// TIA Portal project "Projeto Base" (V17)

(* hardware
DEVICE "S7-1200 station_1"  S7-1200 Station
   slot 0: "Rack_0"  S7-1200 Rack  Rack  V1.0
   slot 1: "PLC_1"  CPU 1212C DC/DC/DC  6ES7 212-1AE40-0XB0  V4.4
DEVICE "HMI_2"  TP700 Comfort
   slot 0: "HMI_2"  TP700 Comfort  6AV2 124-0GC01-0AX0  17.0.0.0
   slot 1: "HMI_RT_2"  TP700 Comfort  6AV2 124-0GC01-0AX0  17.0.0.0
   slot 5: "HMI_2.IE_CP_1"  PROFINET Interface  17.0.0.0
      slot 1: "PROFINET Interface_1"  PROFINET Interface
         slot 1: "Port_1"  Port
         slot 2: "Port_2"  Port
   slot 7: "HMI_2.MPI/DP_CP_1"  MPI/DP Interface  17.0.0.0
*)

// ===== PLC "PLC_1"  CPU 1212C DC/DC/DC =====

VAR_GLOBAL   // PLC tag table "Default tag table"
   "andar_tela" AT %I0.0 : Bool;
   "reset" AT %M0.0 : Bool;
   "voltar_tela" AT %I0.3 : Bool;
   "ligar_led" AT %M0.1 : Bool;
   "led" AT %Q0.0 : Bool;
END_VAR

DATA_BLOCK "DB_IHM"   // DB1
{ S7_Optimized_Access := 'TRUE' }
VERSION : 0.1
   VAR
      IHM_Screen : Array[0..4] of UInt;
      Set_tela : UInt;
      ligar_led : Bool;
   END_VAR
BEGIN
END_DATA_BLOCK

// folder: System blocks/Program resources

DATA_BLOCK "IEC_Counter_0_DB_1"   // DB3
{ S7_Optimized_Access := 'TRUE' }
AUTHOR : Simatic
FAMILY : IEC
NAME : CNTR
VERSION : 1.0
// stored: InstanceOfName IEC_COUNTER
"IEC_COUNTER"
BEGIN
END_DATA_BLOCK

// folder: (top level)

ORGANIZATION_BLOCK "Main"   // OB1, LAD, ProgramCycle
TITLE = "Main Program Sweep (Cycle)"
{ S7_Optimized_Access := 'TRUE' }
VERSION : 0.1
   VAR_INPUT
      Initial_Call : Bool;   // Initial call of this OB
      Remanence : Bool;   // =True, if remanent data are available
   END_VAR
BEGIN

REGION Network 1
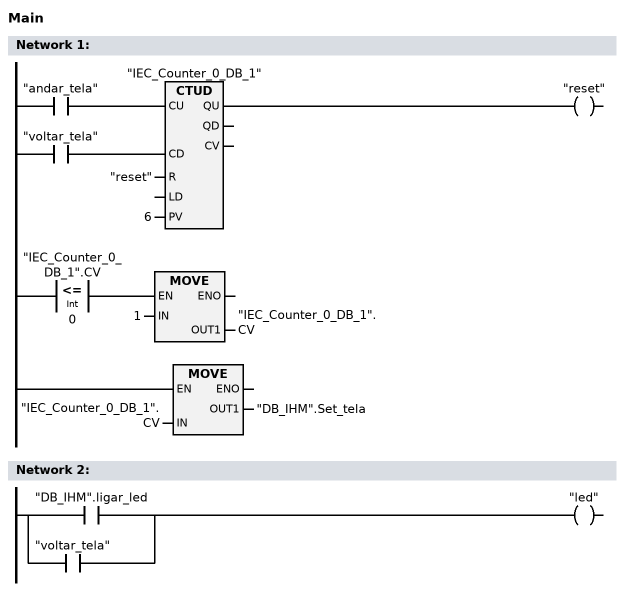
   "IEC_Counter_0_DB_1".CTUD(CU := "andar_tela", CD := "voltar_tela", R := "reset", PV := 6);
   "reset" := "IEC_Counter_0_DB_1".QU;
   IF "IEC_Counter_0_DB_1".CV <= 0 THEN "IEC_Counter_0_DB_1".CV := 1; END_IF;
   "DB_IHM".Set_tela := "IEC_Counter_0_DB_1".CV;
END_REGION

REGION Network 2
   RUNG wire#powerrail
      Contact( "DB_IHM".ligar_led )
      wire#w1
      Coil( "led" )
   END_RUNG
   RUNG wire#powerrail
      Contact( "voltar_tela" )
   END_RUNG wire#w1
   // the same network as SCL:
   "led" := "DB_IHM".ligar_led OR "voltar_tela";
END_REGION
END_ORGANIZATION_BLOCK

(* ===== HMI "HMI_RT_2" =====
system functions are stored by id; their names below are inferred from use
connection "HMI_Connection_2": ETHERNET, S7_1200_OMS

HMI tags "Default tag table"
   "Tag_ScreenNumber" : UInt, internal
   "Numero da tela" : UInt, internal
   "mudarTela" : UInt = PLC DB_IHM.Set_tela AT %DB1.DBW0, 1 s
      on ChangeValue: ActivateScreenByNumber("mudarTela", 0)
   "ligar_led" : Bool = PLC DB_IHM.ligar_led AT %DB1.DBX0.0, 1 s
   "desligar_led" : Bool = PLC DB_IHM.ligar_led AT %M0.1, 1 s
   "ligar_led_interno" : Bool AT %DB1.DBX0.0

screen "Root screen" 800x420, template "Template_1"
   on GenerateScreen: SetTag("Tag_ScreenNumber", 1)
   TextField "HmiScreenItemData" at 65,42 size 640x25; Text 'Welcome to HMI_2 (TP700 Comfort)!'
   Button "Button_1" at 140,160 size 96x32; TextOff 'Ligar Led'
      on Press: function_b3f726e6("ligar_led", 0)
   Button "Button_2" at 255,160 size 146x32; TextOff 'Desligar Led'
      on Click: ResetBit("desligar_led")
      on Press: ResetBit("ligar_led")
   Circle "Circle_1" at 219,218 size 61x61
      Appearance <- "ligar_led"
   IOField "I/O field_1" at 423,160 size 96x32; FormatPattern 1
      ProcessValue <- "ligar_led"

Template "Template_1" 800x420
   Button "Exit" at 720,360 size 78x58; TextOff 'Exit'; PictureOff "ExitRuntime_TP700_Comfort_TR"; PictureOn "ExitRuntime_TP700_Comfort_TR"
      on Release: StopRuntime(0)
   TextField "Template_Text field_1" at 349,115 size 62x23; Text 'Tela 1'
   Button "Start screen_1" at 126,360 size 132x58; TextOn 'Start screen'; TextOff 'CARREGADOR'; PictureOn "NavigateHome_TP700_Comfort_TR"; PictureOff "NavigateHome_TP700_Comfort_TR"
      on Release: ActivateScreen("Root screen", 0)
      on Click: ActivateScreen("Screen_1", 0)
   Button "Start screen" at 1,360 size 116x58; TextOff 'TOPOLOGIA'; TextOn 'Start screen'; PictureOff "NavigateHome_TP700_Comfort_TR"; PictureOn "NavigateHome_TP700_Comfort_TR"
      on Release: ActivateScreen("Root screen", 0)

screen "Screen_1" 800x420
   Button "Button_1" at 142,142 size 96x32; TextOff 'Text'
      on Click: ActivateScreen("Root screen", 0)
   IOField "I/O field_1" at 433,142 size 96x32; FormatPattern 9
      ProcessValue <- "mudarTela"
   TextField "Text field_1" at 309,47 size 62x23; Text 'Tela 2'

screen "Screen_2" 800x420
   TextField "Text field_1" at 372,139 size 62x23; Text 'Tela 3'

screen "Screen_3" 800x420
   TextField "Text field_1" at 352,161 size 62x23; Text 'Tela 4'

screen "Screen_4" 800x420
   TextField "Text field_1" at 372,139 size 62x23; Text 'Tela 5'
*)